// TIA Portal project "Parking" (V15.1)

(* hardware
DEVICE "S71500/ET200MP station_1"  S7-1500 station
   slot 0: "Rail_0"  Rack  6ES7 590-1***0-0AA0
   slot 1: "PLC_1"  CPU 1511TF-1 PN  6ES7 511-1UK01-0AB0  V2.6
      slot 3: "CPU display_1"  6ES7591-1AA00-0AA0
DEVICE "HMI_1"  TP1200 Comfort
   slot 0: "HMI_1"  TP1200 Comfort  6AV2 124-0MC01-0AX0  15.1.0.0
   slot 1: "HMI_RT_1"  TP1200 Comfort  6AV2 124-0MC01-0AX0  15.1.0.0
   slot 5: "HMI_1.IE_CP_1"  PROFINET Interface  15.0.1.0
      slot 1: "PROFINET Interface_1"  PROFINET Interface
         slot 1: "Port_1"  Port
         slot 2: "Port_2"  Port
   slot 7: "HMI_1.MPI/DP_CP_1"  MPI/DP Interface  15.0.1.0
*)

// ===== PLC "PLC_1"  CPU 1511TF-1 PN =====

VAR_GLOBAL   // PLC tag table "Default tag table"
   "Tag_1" AT %I0.1 : Bool;
   "Tag_2" AT %Q0.1 : Bool;
   "System_Byte" AT %MB10000 : Byte;
   "FirstScan" AT %M10000.0 : Bool;
   "DiagStatusUpdate" AT %M10000.1 : Bool;
   "AlwaysTRUE" AT %M10000.2 : Bool;
   "AlwaysFALSE" AT %M10000.3 : Bool;
   "Clock_Byte" AT %MB10010 : Byte;
   "Clock_10Hz" AT %M10010.0 : Bool;
   "Clock_5Hz" AT %M10010.1 : Bool;
   "Clock_2.5Hz" AT %M10010.2 : Bool;
   "Clock_2Hz" AT %M10010.3 : Bool;
   "Clock_1.25Hz" AT %M10010.4 : Bool;
   "Clock_1Hz" AT %M10010.5 : Bool;
   "Clock_0.625Hz" AT %M10010.6 : Bool;
   "Clock_0.5Hz" AT %M10010.7 : Bool;
END_VAR

DATA_BLOCK "Blok_funkcyjny"   // DB1
{ S7_Optimized_Access := 'TRUE' }
VERSION : 0.1
// stored: InstanceOfName Funkcja1
"Funkcja1"
BEGIN
END_DATA_BLOCK

DATA_BLOCK "Blok danych"   // DB2
{ S7_Optimized_Access := 'TRUE' }
VERSION : 0.1
   VAR
      otworz : Bool;
      zamknij : Bool;
      stan_otwarcia_bramy : Bool;
      brama : Real := 0.01;
      polozenie_bramy : Real;
      polozenie_bramy_int : Int;
      impulsy : Bool;
      zb_narast : Bool;
      zb_opad : Bool;
      generator1Hz : Bool;
      ograniczenie_max : Real := 100.0;
      ograniczenie_min : Int := 0;
      przerwij : Bool;
      przerwij1 : Bool;
      przejazd_mozliwy : Bool;
      przejazd_niemozliwy : Bool;
      rejestracje : Array[0..20] of String;
      random_rejestracja : String := 'Wpisz';
      pozwolenie : Bool;
      licznik : Int;
      wpuszczenie : Bool;
      sprawdz_czy_wpuscic : Bool;
      samochod_podjechal : Bool;
      check_again : Bool;
      probne : Bool;
      samochod_spoza_listy : Bool;
      Automatyczne_zamkniecie : Time := T#15s;
      otworz_automat : Bool;
      zamknij_automat : Bool;
      przejazd_mozliwy1 : Bool;
      przejazd_niemozliwy1 : Bool;
      wlacz : Bool;
      wylacz : Bool;
      zalacz : Bool;
      podglad_rejestracji : Bool;
      dodaj_rejestracje_do_bazy : Bool;
      numer_do_bazy : Int;
      dodaj_do_bazy : String;
      procent : Real;
   END_VAR
BEGIN
   rejestracje[0] := 'TKI0';
   rejestracje[1] := 'TKI1';
   rejestracje[2] := 'TKI2';
   rejestracje[3] := 'TKI3';
END_DATA_BLOCK

DATA_BLOCK "Sprawdzanie_rejestracji_DB"   // DB3
{ S7_Optimized_Access := 'TRUE' }
VERSION : 0.1
// stored: InstanceOfName Sprawdzanie_rejestracji
"Sprawdzanie_rejestracji"
BEGIN
   random_rejestracja := 'Wpisz';
END_DATA_BLOCK

// folder: System blocks/Program resources

DATA_BLOCK "IEC_Timer_0_DB"   // DB4
{ S7_Optimized_Access := 'TRUE' }
AUTHOR : Simatic
FAMILY : IEC
NAME : IEC_TMR
VERSION : 1.0
// stored: InstanceOfName IEC_TIMER
"IEC_TIMER"
BEGIN
END_DATA_BLOCK

// folder: (top level)

FUNCTION_BLOCK "Funkcja1"   // FB1, LAD
{ S7_Optimized_Access := 'TRUE' }
VERSION : 0.1
   VAR_INPUT
      otworz : Bool;
      zamknij : Bool;
   END_VAR
   VAR_OUTPUT
      przejazd_niemozliwy : Bool;
      przejazd_mozliwy : Bool;
      procent : Int;
   END_VAR
   VAR
      przerwij : Bool;
      przerwij1 : Bool;
      stan_otwarcia_bramy : Bool;
      polozenie_bramy : Real;
      brama : Real := 0.01;
      polozenie_bramy_int : Int;
      licznik : Int;
   END_VAR
   VAR CONSTANT
      ograniczenie_min : Int;
      ograniczenie_max : Int := 100;
   END_VAR
   VAR_TEMP   // added for the SCL form of the ladder/FBD networks
      _w1 : Bool;
      _w2 : Bool;
   END_VAR
BEGIN

REGION Network 1
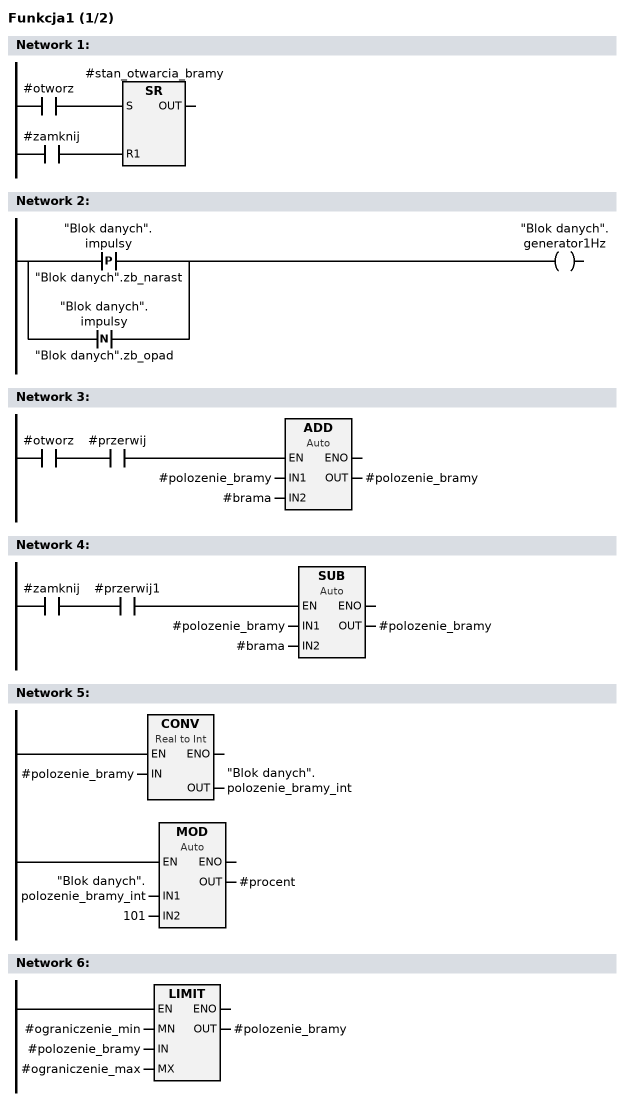
   RUNG wire#powerrail
      Contact( #otworz )
      S_SR(operand := #stan_otwarcia_bramy, r1 := wire#w1)
   END_RUNG
   RUNG wire#powerrail
      Contact( #zamknij )
   END_RUNG wire#w1
   // the same network as SCL:
   IF #otworz THEN
       #stan_otwarcia_bramy := TRUE;   // SR flip-flop
   END_IF;
   IF #zamknij THEN #stan_otwarcia_bramy := FALSE; END_IF;
END_REGION

REGION Network 2
   RUNG wire#powerrail
      P_Contact(operand := "Blok danych".impulsy, bit := "Blok danych".zb_narast)
      wire#w1
      Coil( "Blok danych".generator1Hz )
   END_RUNG
   RUNG wire#powerrail
      N_Contact(operand := "Blok danych".impulsy, bit := "Blok danych".zb_opad)
   END_RUNG wire#w1
   // the same network as SCL:
   #_w1 := "Blok danych".impulsy AND NOT "Blok danych".zb_narast;   // rising edge of "Blok danych".impulsy
   "Blok danych".zb_narast := "Blok danych".impulsy;
   #_w2 := NOT "Blok danych".impulsy AND "Blok danych".zb_opad;   // falling edge of "Blok danych".impulsy
   "Blok danych".zb_opad := "Blok danych".impulsy;
   "Blok danych".generator1Hz := #_w1 OR #_w2;
END_REGION

REGION Network 3
   RUNG wire#powerrail
      Contact( #otworz )
      Contact( #przerwij )
      Add(in1 := #polozenie_bramy, in2 := #brama, out => #polozenie_bramy)
   END_RUNG
   // the same network as SCL:
   IF #otworz AND #przerwij THEN #polozenie_bramy := #polozenie_bramy + #brama; END_IF;
END_REGION

REGION Network 4
   RUNG wire#powerrail
      Contact( #zamknij )
      Contact( #przerwij1 )
      Sub(in1 := #polozenie_bramy, in2 := #brama, out => #polozenie_bramy)
   END_RUNG
   // the same network as SCL:
   IF #zamknij AND #przerwij1 THEN #polozenie_bramy := #polozenie_bramy - #brama; END_IF;
END_REGION

REGION Network 5
   RUNG wire#powerrail
      { S7_Templates := "[SrcType := Real, DestType := Int]" } Convert(in := #polozenie_bramy, out => "Blok danych".polozenie_bramy_int)
   END_RUNG
   RUNG wire#powerrail
      Mod(in1 := "Blok danych".polozenie_bramy_int, in2 := 101, out => #procent)
   END_RUNG
   // the same network as SCL:
   "Blok danych".polozenie_bramy_int := REAL_TO_INT(#polozenie_bramy);
   #procent := "Blok danych".polozenie_bramy_int MOD 101;
END_REGION

REGION Network 6
   #polozenie_bramy := LIMIT(MN := #ograniczenie_min, IN := #polozenie_bramy, MX := #ograniczenie_max);
END_REGION

REGION Network 7
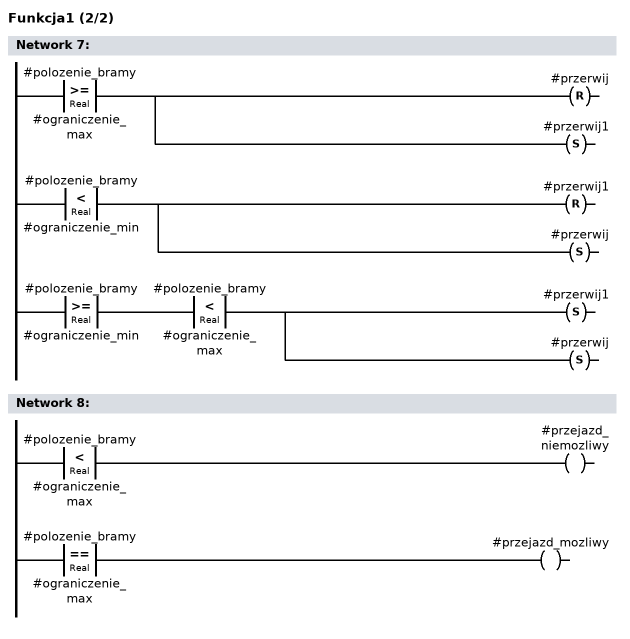
   RUNG wire#powerrail
      { S7_Templates := "SrcType := Real" } GE_Contact(in1 := #polozenie_bramy, in2 := #ograniczenie_max)
      wire#w1
      R_Coil( #przerwij )
   END_RUNG
   RUNG wire#w1
      S_Coil( #przerwij1 )
   END_RUNG
   RUNG wire#powerrail
      { S7_Templates := "SrcType := Real" } LT_Contact(in1 := #polozenie_bramy, in2 := #ograniczenie_min)
      wire#w2
      R_Coil( #przerwij1 )
   END_RUNG
   RUNG wire#w2
      S_Coil( #przerwij )
   END_RUNG
   RUNG wire#powerrail
      { S7_Templates := "SrcType := Real" } GE_Contact(in1 := #polozenie_bramy, in2 := #ograniczenie_min)
      { S7_Templates := "SrcType := Real" } LT_Contact(in1 := #polozenie_bramy, in2 := #ograniczenie_max)
      wire#w3
      S_Coil( #przerwij1 )
   END_RUNG
   RUNG wire#w3
      S_Coil( #przerwij )
   END_RUNG
   // the same network as SCL:
   IF #polozenie_bramy >= #ograniczenie_max THEN
       #przerwij := FALSE;
       #przerwij1 := TRUE;
   END_IF;
   IF #polozenie_bramy < #ograniczenie_min THEN
       #przerwij1 := FALSE;
       #przerwij := TRUE;
   END_IF;
   IF (#polozenie_bramy >= #ograniczenie_min) AND (#polozenie_bramy < #ograniczenie_max) THEN
       #przerwij1 := TRUE;
       #przerwij := TRUE;
   END_IF;
END_REGION

REGION Network 8
   RUNG wire#powerrail
      { S7_Templates := "SrcType := Real" } LT_Contact(in1 := #polozenie_bramy, in2 := #ograniczenie_max)
      Coil( #przejazd_niemozliwy )
   END_RUNG
   RUNG wire#powerrail
      { S7_Templates := "SrcType := Real" } EQ_Contact(in1 := #polozenie_bramy, in2 := #ograniczenie_max)
      Coil( #przejazd_mozliwy )
   END_RUNG
   // the same network as SCL:
   #przejazd_niemozliwy := #polozenie_bramy < #ograniczenie_max;
   #przejazd_mozliwy := #polozenie_bramy = #ograniczenie_max;
END_REGION
END_FUNCTION_BLOCK

FUNCTION_BLOCK "Sprawdzanie_rejestracji"   // FB2, LAD
{ S7_Optimized_Access := 'TRUE' }
VERSION : 0.1
   VAR_INPUT
      random_rejestracja : String;
      sprawdz_czy_wpuscic : Bool;
      Nie_ma_sprawdz_again : Bool;
      zezwol_spoza_listy : Bool;
      nowa_rejestracja : String;
      numer_w_bazie : Int;
      dodaj_rejestracje_do_bazy : Bool;
   END_VAR
   VAR_OUTPUT
      pozwolenie_na_przejazd : Bool;
   END_VAR
   VAR
      licznik : Int;
      limit_inkrementu : Bool;
      probne : Bool;
      probne2 : Bool;
      dodawanie_rejestracji : Bool;
   END_VAR
   VAR CONSTANT
      "ilosc rejestracji min" : Int;
      "ilosc rejestracji max" : Int := 20;
      "wylaczenie sprawdzania" : Int := 3;
      "wylaczenie sprawdzania2" : Int := 100;
   END_VAR
BEGIN

REGION Network 1
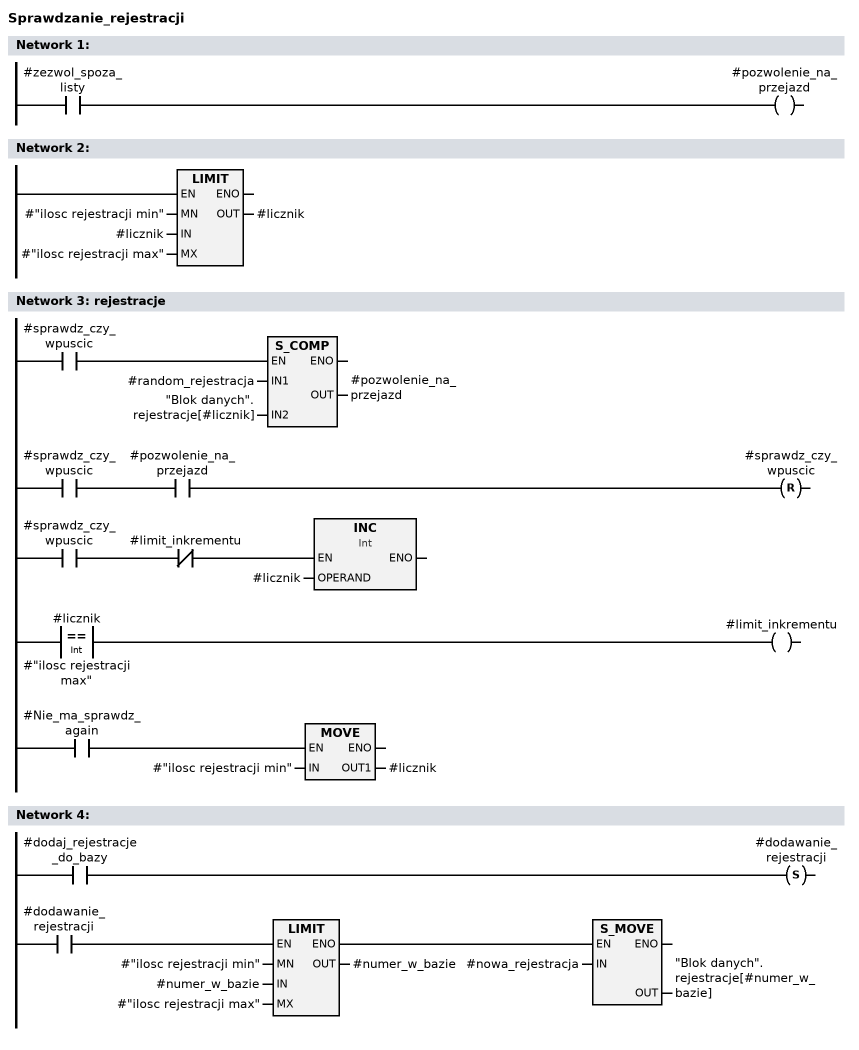
   RUNG wire#powerrail
      Contact( #zezwol_spoza_listy )
      Coil( #pozwolenie_na_przejazd )
   END_RUNG
   // the same network as SCL:
   #pozwolenie_na_przejazd := #zezwol_spoza_listy;
END_REGION

REGION Network 2
   #licznik := LIMIT(MN := #"ilosc rejestracji min", IN := #licznik, MX := #"ilosc rejestracji max");
END_REGION

REGION Network 3: rejestracje
   IF #sprawdz_czy_wpuscic THEN
       S_COMP(IN1 := #random_rejestracja,
              IN2 := "Blok danych".rejestracje[#licznik],
              OUT => #pozwolenie_na_przejazd);
   END_IF;
   IF #sprawdz_czy_wpuscic AND #pozwolenie_na_przejazd THEN #sprawdz_czy_wpuscic := FALSE; END_IF;
   IF #sprawdz_czy_wpuscic AND NOT #limit_inkrementu THEN #licznik := #licznik + 1; END_IF;
   #limit_inkrementu := #licznik = #"ilosc rejestracji max";
   IF #Nie_ma_sprawdz_again THEN #licznik := #"ilosc rejestracji min"; END_IF;
END_REGION

REGION Network 4
   IF #dodaj_rejestracje_do_bazy THEN #dodawanie_rejestracji := TRUE; END_IF;
   IF #dodawanie_rejestracji THEN
       #numer_w_bazie := LIMIT(MN := #"ilosc rejestracji min", IN := #numer_w_bazie, MX := #"ilosc rejestracji max");
       "Blok danych".rejestracje[#numer_w_bazie] := #nowa_rejestracja;
   END_IF;
END_REGION
END_FUNCTION_BLOCK

ORGANIZATION_BLOCK "Main"   // OB1, LAD, ProgramCycle
TITLE = "Main Program Sweep (Cycle)"
{ S7_Optimized_Access := 'TRUE' }
VERSION : 0.1
   VAR_INPUT
      Initial_Call : Bool;   // Initial call of this OB
      Remanence : Bool;   // =True, if remanent data are available
   END_VAR
   VAR_TEMP   // added for the SCL form of the ladder/FBD networks
      _w1 : Bool;
   END_VAR
BEGIN

REGION Network 1
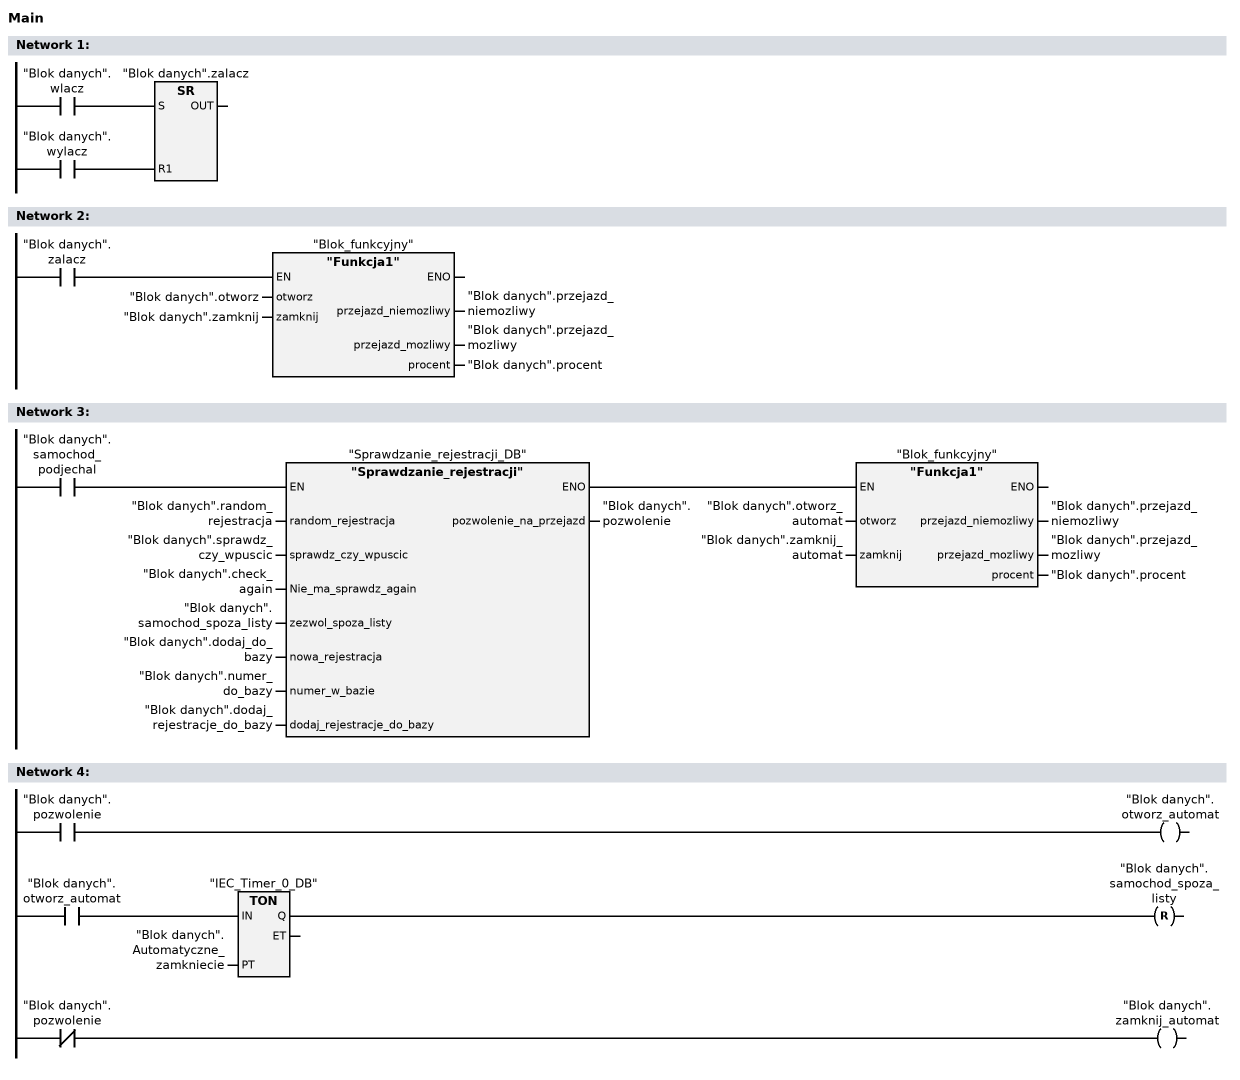
   RUNG wire#powerrail
      Contact( "Blok danych".wlacz )
      S_SR(operand := "Blok danych".zalacz, r1 := wire#w1)
   END_RUNG
   RUNG wire#powerrail
      Contact( "Blok danych".wylacz )
   END_RUNG wire#w1
   // the same network as SCL:
   IF "Blok danych".wlacz THEN
       "Blok danych".zalacz := TRUE;   // SR flip-flop
   END_IF;
   IF "Blok danych".wylacz THEN "Blok danych".zalacz := FALSE; END_IF;
END_REGION

REGION Network 2
   RUNG wire#powerrail
      Contact( "Blok danych".zalacz )
      "Blok_funkcyjny"(otworz := "Blok danych".otworz, zamknij := "Blok danych".zamknij, przejazd_niemozliwy => "Blok danych".przejazd_niemozliwy, przejazd_mozliwy => "Blok danych".przejazd_mozliwy, procent => "Blok danych".procent)
   END_RUNG
   // the same network as SCL:
   IF "Blok danych".zalacz THEN
       "Blok_funkcyjny"(otworz := "Blok danych".otworz,   // "Funkcja1"
                        zamknij := "Blok danych".zamknij,
                        przejazd_niemozliwy => "Blok danych".przejazd_niemozliwy,
                        przejazd_mozliwy => "Blok danych".przejazd_mozliwy,
                        procent => "Blok danych".procent);
   END_IF;
END_REGION

REGION Network 3
   RUNG wire#powerrail
      Contact( "Blok danych".samochod_podjechal )
      "Sprawdzanie_rejestracji_DB"(random_rejestracja := "Blok danych".random_rejestracja, sprawdz_czy_wpuscic := "Blok danych".sprawdz_czy_wpuscic, Nie_ma_sprawdz_again := "Blok danych".check_again, zezwol_spoza_listy := "Blok danych".samochod_spoza_listy, nowa_rejestracja := "Blok danych".dodaj_do_bazy, numer_w_bazie := "Blok danych".numer_do_bazy, dodaj_rejestracje_do_bazy := "Blok danych".dodaj_rejestracje_do_bazy, pozwolenie_na_przejazd => "Blok danych".pozwolenie)
      "Blok_funkcyjny"(otworz := "Blok danych".otworz_automat, zamknij := "Blok danych".zamknij_automat, przejazd_niemozliwy => "Blok danych".przejazd_niemozliwy, przejazd_mozliwy => "Blok danych".przejazd_mozliwy, procent => "Blok danych".procent)
   END_RUNG
   // the same network as SCL:
   "Sprawdzanie_rejestracji_DB"(EN := "Blok danych".samochod_podjechal,   // "Sprawdzanie_rejestracji"
                           random_rejestracja := "Blok danych".random_rejestracja,
                           sprawdz_czy_wpuscic := "Blok danych".sprawdz_czy_wpuscic,
                           Nie_ma_sprawdz_again := "Blok danych".check_again,
                           zezwol_spoza_listy := "Blok danych".samochod_spoza_listy,
                           nowa_rejestracja := "Blok danych".dodaj_do_bazy,
                           numer_w_bazie := "Blok danych".numer_do_bazy,
                           dodaj_rejestracje_do_bazy := "Blok danych".dodaj_rejestracje_do_bazy,
                           pozwolenie_na_przejazd => "Blok danych".pozwolenie,
                           ENO => #_w1);
   IF #_w1 THEN
       "Blok_funkcyjny"(otworz := "Blok danych".otworz_automat,   // "Funkcja1"
                        zamknij := "Blok danych".zamknij_automat,
                        przejazd_niemozliwy => "Blok danych".przejazd_niemozliwy,
                        przejazd_mozliwy => "Blok danych".przejazd_mozliwy,
                        procent => "Blok danych".procent);
   END_IF;
END_REGION

REGION Network 4
   "Blok danych".otworz_automat := "Blok danych".pozwolenie;
   "IEC_Timer_0_DB".TON(IN := "Blok danych".otworz_automat, PT := "Blok danych".Automatyczne_zamkniecie);
   IF "IEC_Timer_0_DB".Q THEN "Blok danych".samochod_spoza_listy := FALSE; END_IF;
   "Blok danych".zamknij_automat := NOT "Blok danych".pozwolenie;
END_REGION
END_ORGANIZATION_BLOCK

ORGANIZATION_BLOCK "Generator1Hz"   // OB30, LAD, CyclicInterrupt
{ S7_Optimized_Access := 'TRUE' }
VERSION : 0.1
   VAR_INPUT
      Initial_Call : Bool;   // Initial call of this OB
      Event_Count : Int;   // Events discarded
   END_VAR
BEGIN

REGION Network 1
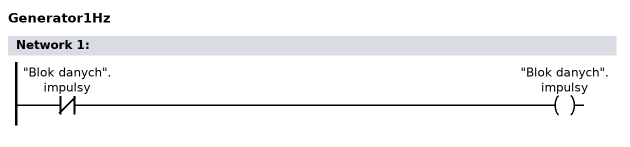
   RUNG wire#powerrail
      I_Contact( "Blok danych".impulsy )
      Coil( "Blok danych".impulsy )
   END_RUNG
   // the same network as SCL:
   "Blok danych".impulsy := NOT "Blok danych".impulsy;
END_REGION
END_ORGANIZATION_BLOCK

(* ===== HMI "HMI_RT_1" =====
system functions are stored by id; their names below are inferred from use
connection "HMI_Connection_1": ETHERNET, S7_1500_OMS

HMI tags "Default tag table"
   "Tag_ScreenNumber" : UInt, internal
   "Blok danych_polozenie_bramy" : Real = PLC "Blok danych".polozenie_bramy, 1 s
   "Blok danych_polozenie_bramy_int" : Int = PLC "Blok danych".polozenie_bramy_int, 1 s
   "Blok danych_przejazd_mozliwy" : Bool = PLC "Blok danych".przejazd_mozliwy, 1 s
   "Blok danych_przejazd_niemozliwy" : Bool = PLC "Blok danych".przejazd_niemozliwy, 1 s
   "Blok danych_otworz" : Bool = PLC "Blok danych".otworz, 1 s
   "Blok danych_zamknij" : Bool = PLC "Blok danych".zamknij, 1 s
   "Blok_funkcyjny_polozenie_bramy_int" : Int = PLC Blok_funkcyjny.polozenie_bramy_int, 1 s
   "Blok_funkcyjny_przejazd_mozliwy" : Bool = PLC Blok_funkcyjny.przejazd_mozliwy, 1 s
   "Blok_funkcyjny_przejazd_niemozliwy" : Bool = PLC Blok_funkcyjny.przejazd_niemozliwy, 1 s
   "Blok_funkcyjny_otworz" : Bool = PLC Blok_funkcyjny.otworz, 1 s
   "Blok_funkcyjny_zamknij" : Bool = PLC Blok_funkcyjny.zamknij, 1 s
   "Blok danych_rejestracje" : Array [0..20] of String[254] = PLC "Blok danych".rejestracje, 1 s
   "Blok danych_rejestracje{0}" : String[254] = PLC "Blok danych".rejestracje[0], 1 s
   "Blok danych_samochod_spoza_listy" : Bool = PLC "Blok danych".samochod_spoza_listy, 1 s
   "Blok danych_dodaj_rejestracje_do_bazy" : Bool = PLC "Blok danych".dodaj_rejestracje_do_bazy, 1 s
   "Blok danych_numer_do_bazy" : Int = PLC "Blok danych".numer_do_bazy, 1 s
   "Blok danych_dodaj_do_bazy" : String[254] = PLC "Blok danych".dodaj_do_bazy, 1 s
   "Blok danych_procent" : Real = PLC "Blok danych".procent, 1 s
   "Blok danych_samochod_podjechal" : Bool = PLC "Blok danych".samochod_podjechal, 1 s
   "Blok danych_random_rejestracja" : String[254] = PLC "Blok danych".random_rejestracja, 1 s
   "Blok danych_sprawdz_czy_wpuscic" : Bool = PLC "Blok danych".sprawdz_czy_wpuscic, 1 s
   "Blok danych_check_again" : Bool = PLC "Blok danych".check_again, 1 s
   "Blok danych_wlacz" : Bool = PLC "Blok danych".wlacz, 1 s
   "Blok danych_wylacz" : Bool = PLC "Blok danych".wylacz, 1 s

screen "Root screen" 1280x740, template "Template_1"
   on GenerateScreen: SetTag("Tag_ScreenNumber", 1)
   TextField "HmiScreenItemData_3" at 124,29 size 1024x27; Text 'Obsluga parkingu'
   Button "HmiScreenItemData" at 36,36 size 159x47; TextOff 'Ekran administracyjny'; PictureOff "Navigates to Ekran administracyjny for TP1200 Comfort 15.1.0.0"; PictureOn "Navigates to Ekran administracyjny for TP1200 Comfort 15.1.0.0"
      on Release: ActivateScreen("Ekran administracyjny", 0)
   Button "HmiScreenItemData_1" at 36,95 size 159x47; TextOff 'Ekran wjazdowy'; PictureOff "Navigates to Ekran wjazdowy for TP1200 Comfort 15.1.0.0"; PictureOn "Navigates to Ekran wjazdowy for TP1200 Comfort 15.1.0.0"
      on Release: ActivateScreen("Ekran wjazdowy", 0)
   Button "HmiScreenItemData_2" at 36,154 size 159x47; TextOff 'Ekran wyjazdowy'; PictureOff "Navigates to Ekran wyjazdowy for TP1200 Comfort 15.1.0.0"; PictureOn "Navigates to Ekran wyjazdowy for TP1200 Comfort 15.1.0.0"
      on Release: ActivateScreen("Ekran wyjazdowy", 0)
   Switch "Switch_1" at 437,99 size 120x88; CaptionText 'Switch'; TextOff 'Zalacz'; TextOn 'ON'
      ProcessValue <- "Blok danych_wlacz"
   Switch "Switch_2" at 799,99 size 120x88; CaptionText 'Switch'; TextOff 'Wylacz'; TextOn 'ON'
      ProcessValue <- "Blok danych_wylacz"

Template "Template_1" 1280x740
   Button "Exit" at 1200,679 size 78x59; TextOff 'Exit'; PictureOff "ExitRuntime_TP1200_Comfort_TR"; PictureOn "ExitRuntime_TP1200_Comfort_TR"
      on Release: StopRuntime(0)
   Button "Template_Button" at 1120,679 size 78x59; TextOff 'Text'
   Button "Template_Button_1" at 1040,679 size 78x59; TextOff 'Text'
   Button "Template_Button_2" at 960,679 size 78x59; TextOff 'Text'
   Button "Template_Button_3" at 880,679 size 78x59; TextOff 'Text'
   Button "Template_Button_4" at 800,679 size 78x59; TextOff 'Text'
   Button "Template_Button_5" at 720,679 size 78x59; TextOff 'Text'
   Button "Template_Button_6" at 640,679 size 78x59; TextOff 'Text'
   Button "Template_Button_7" at 561,679 size 78x59; TextOff 'Text'
   Button "Template_Button_8" at 481,679 size 78x59; TextOff 'Text'
   Button "Template_Button_9" at 401,679 size 78x59; TextOff 'Text'
   Button "Template_Button_10" at 321,679 size 78x59; TextOff 'Text'
   Button "Template_Button_11" at 241,679 size 78x59; TextOff 'Text'
   Button "Log on" at 161,679 size 78x59; TextOff 'Log on'; PictureOff "Login_TP1200_Comfort_TR"; PictureOn "Login_TP1200_Comfort_TR"
      on Release: function_a2a04561()
   Button "Alarms" at 81,679 size 78x59; TextOff 'Alarms'; PictureOff "AlarmDisplay_TP1200_Comfort_TR"; PictureOn "AlarmDisplay_TP1200_Comfort_TR"
      on Release: function_ef3f5d25("Alarm window_Unacknowledged", -1)
   Button "Start screen" at 1,679 size 78x59; TextOff 'Start screen'; PictureOff "NavigateHome_TP1200_Comfort_TR"; PictureOn "NavigateHome_TP1200_Comfort_TR"
      on Release: ActivateScreen("Root screen", 0)

screen "Ekran administracyjny" 1280x740, template "Template_1"
   on GenerateScreen: SetTag("Tag_ScreenNumber", 2)
   Button "Back" at 1,1 size 159x47; TextOff 'Back'
      on Release: ActivateScreen("Root screen", 0)
   Rectangle "Rectangle_3" at 70,167 size 243x23
      HorizontalMovement <- "Blok danych_polozenie_bramy_int"
   Circle "Circle_1" at 620,189 size 68x68
      Appearance <- "Blok danych_przejazd_mozliwy"
   Circle "Circle_2" at 811,191 size 66x66
      Appearance <- "Blok danych_przejazd_niemozliwy"
   TextField "Text field_1" at 572,165 size 170x25; Text 'Przejazd mozliwy'
   TextField "Text field_2" at 760,166 size 199x25; Text 'Przejazd niemozliwy'
   Switch "Switch_1" at 590,50 size 120x88; CaptionText 'Switch'; TextOff 'Otworz'; TextOn 'Otwieranie'
      ProcessValue <- "Blok danych_otworz"
   Switch "Switch_2" at 795,49 size 120x88; TextOn 'Zamykanie'; CaptionText 'Switch'; TextOff 'Zamknij'
      ProcessValue <- "Blok danych_zamknij"
   Button "Button_1" at 67,85 size 278x32; TextOff 'Zobacz liste zezwolonych aut'
      on Click: ActivateScreen("Lista_zezwolonych", 0)
   TextField "Text field_3" at 455,398 size 250x25; Text 'Stan otwarcia bramy w %'
   Bar "Bar_1" at 541,424 size 80x230; MinimumValue 0; MaximumValue 100
      ProcessValue <- "Blok danych_procent"
   TextField "Text field_4" at 787,281 size 493x25; Text 'Jezeli samochod podjechal wcisnij przycisk ponizej'
   TextField "Text field_5" at 947,370 size 215x25; Text 'Podaj rejestracje auta'
   IOField "I/O field_1" at 980,395 size 96x32; FormatPattern ????????????????????????????????????????????????????????????????????????????????
      ProcessValue <- "Blok danych_random_rejestracja"
   TextField "Text field_6" at 914,437 size 271x25; Text 'Sprawdz czy ma pozwolenie'
   Switch "Switch_3" at 980,308 size 106x60; CaptionText 'Switch'; TextOff 'OFF'; TextOn 'ON'
      ProcessValue <- "Blok danych_samochod_podjechal"
   Switch "Switch_4" at 980,460 size 120x55; CaptionText 'Switch'; TextOff 'OFF'; TextOn 'ON'
      ProcessValue <- "Blok danych_sprawdz_czy_wpuscic"
   Switch "Switch_5" at 969,622 size 120x51; CaptionText 'Switch'; TextOff 'OFF'; TextOn 'ON'
      ProcessValue <- "Blok danych_samochod_spoza_listy"
   TextField "Text field_7" at 950,586 size 163x25; Text 'Zezwol na wjazd'
   Button "Button_2" at 716,540 size 560x32; TextOff 'Jezeli auta nie ma na liscie, a chcesz sprawdzic kolejne-kliknij tu'
      on Press: function_b14e0dd5("Blok danych_check_again", 0)

screen "Ekran wjazdowy" 1280x740, template "Template_1"
   on GenerateScreen: SetTag("Tag_ScreenNumber", 3)
   Button "Back" at 1,1 size 159x47; TextOff 'Back'
      on Release: ActivateScreen("Root screen", 0)
   Rectangle "Rectangle_3" at 77,303 size 243x23
      HorizontalMovement <- "Blok danych_polozenie_bramy_int"
   Circle "Circle_1" at 527,219 size 68x68
      Appearance <- "Blok danych_przejazd_mozliwy"
   Circle "Circle_2" at 711,221 size 66x66
      Appearance <- "Blok danych_przejazd_niemozliwy"
   TextField "Text field_1" at 479,186 size 170x25; Text 'Przejazd mozliwy'
   TextField "Text field_2" at 664,186 size 199x25; Text 'Przejazd niemozliwy'

screen "Ekran wyjazdowy" 1280x740, template "Template_1"
   on GenerateScreen: SetTag("Tag_ScreenNumber", 4)
   Button "Back" at 1,1 size 159x47; TextOff 'Back'
      on Release: ActivateScreen("Root screen", 0)
   Rectangle "Rectangle_3" at 29,179 size 243x23
      HorizontalMovement <- "Blok danych_polozenie_bramy_int"
   Circle "Circle_1" at 479,95 size 68x68
      Appearance <- "Blok danych_przejazd_mozliwy"
   Circle "Circle_2" at 663,97 size 66x66
      Appearance <- "Blok danych_przejazd_niemozliwy"
   TextField "Text field_1" at 431,62 size 170x25; Text 'Przejazd mozliwy'
   TextField "Text field_2" at 616,62 size 199x25; Text 'Przejazd niemozliwy'

screen "Lista_zezwolonych" 1280x740
   Button "Button_1" at 29,45 size 96x32; TextOff 'Wroc'
      on Click: ActivateScreen("Ekran administracyjny", 0)
   IOField "I/O field_1" at 67,123 size 96x32; FormatPattern ????????????????????????????????????????????????????????????????????????????????
      ProcessValue <- "[1]"
   IOField "I/O field_2" at 67,155 size 96x32; FormatPattern ????????????????????????????????????????????????????????????????????????????????
      ProcessValue <- "[2]"
   IOField "I/O field_3" at 67,187 size 96x32; FormatPattern ????????????????????????????????????????????????????????????????????????????????
      ProcessValue <- "[3]"
   IOField "I/O field_4" at 67,219 size 96x32; FormatPattern ????????????????????????????????????????????????????????????????????????????????
      ProcessValue <- "[4]"
   IOField "I/O field_5" at 67,251 size 96x32; FormatPattern ????????????????????????????????????????????????????????????????????????????????
      ProcessValue <- "[5]"
   IOField "I/O field_6" at 67,283 size 96x32; FormatPattern ????????????????????????????????????????????????????????????????????????????????
      ProcessValue <- "[6]"
   IOField "I/O field_7" at 67,315 size 96x32; FormatPattern ????????????????????????????????????????????????????????????????????????????????
      ProcessValue <- "[7]"
   IOField "I/O field_8" at 67,347 size 96x32; FormatPattern ????????????????????????????????????????????????????????????????????????????????
      ProcessValue <- "[8]"
   IOField "I/O field_9" at 67,379 size 96x32; FormatPattern ????????????????????????????????????????????????????????????????????????????????
      ProcessValue <- "[9]"
   IOField "I/O field_10" at 67,411 size 96x32; FormatPattern ????????????????????????????????????????????????????????????????????????????????
      ProcessValue <- "[10]"
   IOField "I/O field_11" at 67,443 size 96x32; FormatPattern ????????????????????????????????????????????????????????????????????????????????
      ProcessValue <- "[11]"
   IOField "I/O field_12" at 67,475 size 96x32; FormatPattern ????????????????????????????????????????????????????????????????????????????????
      ProcessValue <- "[12]"
   IOField "I/O field_13" at 67,507 size 96x32; FormatPattern ????????????????????????????????????????????????????????????????????????????????
      ProcessValue <- "[13]"
   IOField "I/O field_14" at 67,539 size 96x32; FormatPattern ????????????????????????????????????????????????????????????????????????????????
      ProcessValue <- "[14]"
   IOField "I/O field_15" at 67,571 size 96x32; FormatPattern ????????????????????????????????????????????????????????????????????????????????
      ProcessValue <- "[15]"
   IOField "I/O field_16" at 67,603 size 96x32; FormatPattern ????????????????????????????????????????????????????????????????????????????????
      ProcessValue <- "[16]"
   IOField "I/O field_17" at 67,635 size 96x32; FormatPattern ????????????????????????????????????????????????????????????????????????????????
      ProcessValue <- "[17]"
   IOField "I/O field_18" at 67,667 size 96x32; FormatPattern ????????????????????????????????????????????????????????????????????????????????
      ProcessValue <- "[18]"
   IOField "I/O field_19" at 67,699 size 96x32; FormatPattern ????????????????????????????????????????????????????????????????????????????????
      ProcessValue <- "[19]"
   IOField "I/O field_20" at 67,91 size 96x32; FormatPattern ????????????????????????????????????????????????????????????????????????????????
      ProcessValue <- "[0]"
   IOField "I/O field_21" at 339,133 size 96x32; FormatPattern s99999
      ProcessValue <- "Blok danych_numer_do_bazy"
   IOField "I/O field_22" at 339,203 size 96x32; FormatPattern ????????????????????????????????????????????????????????????????????????????????
      ProcessValue <- "Blok danych_dodaj_do_bazy"
   TextField "Text field_1" at 208,98 size 509x25; Text 'Podaj numer, pod ktorym umiescisz nowa rejestracje'
   TextField "Text field_2" at 278,170 size 228x25; Text 'Podaj nazwe rejestracji'
   TextField "Text field_3" at 42,91 size 17x25; Text '0'
   TextField "Text field_4" at 42,130 size 17x25; Text '1'
   TextField "Text field_5" at 43,160 size 17x25; Text '2'
   TextField "Text field_6" at 43,192 size 17x25; Text '3'
   TextField "Text field_7" at 43,225 size 17x25; Text '4'
   TextField "Text field_8" at 41,256 size 17x25; Text '5'
   TextField "Text field_9" at 44,290 size 17x25; Text '6'
   TextField "Text field_10" at 44,319 size 17x25; Text '7'
   TextField "Text field_11" at 44,347 size 17x25; Text '8'
   TextField "Text field_12" at 45,384 size 17x25; Text '9'
   TextField "Text field_13" at 35,417 size 29x25; Text '10'
   TextField "Text field_14" at 36,449 size 29x25; Text '11'
   TextField "Text field_15" at 41,482 size 29x25; Text '13'
   TextField "Text field_16" at 40,514 size 29x25; Text '14'
   TextField "Text field_17" at 40,545 size 29x25; Text '15'
   TextField "Text field_18" at 43,576 size 29x25; Text '16'
   TextField "Text field_19" at 40,609 size 29x25; Text '17'
   TextField "Text field_20" at 41,640 size 29x25; Text '18'
   TextField "Text field_21" at 42,672 size 29x25; Text '19'
   TextField "Text field_22" at 35,699 size 29x25; Text '20'
*)